Omron CX-Programmer project NewProject (CX-Programmer 9.73)

# PLC NewPLC1: CP1E N30

## Program NewProgram1 (cyclic task 0)

### Section Section1

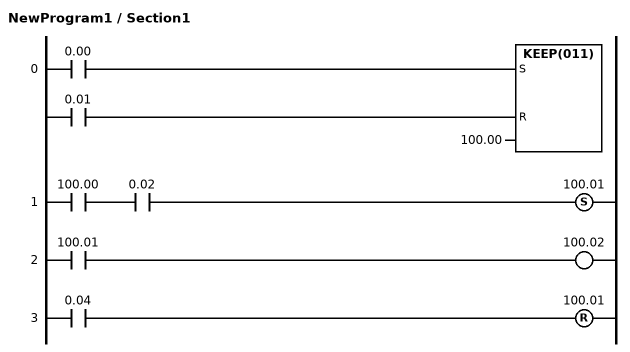
; rung 0
LD 0.00
LD 0.01
KEEP(011) 100.00
; rung 1
LD 100.00
AND 0.02
SET 100.01
; rung 2
LD 100.01
OUT 100.02
; rung 3
LD 0.04
RSET 100.01

### Section END
; rung 0
END(001)